// TIA Portal V18 export
DATA_BLOCK "Axis_FB_DB"   // DB2200
// stored: AutoNumber false, InstanceOfName Axis_FB, InstanceOfType FB
"Axis_FB"
   // VAR RETAIN
   //    IAI_Axis { S7_SetPoint := 'True'} : Array[1..3] of "IAI_BASE_FB";
   // END_VAR
BEGIN
   // IAI_Axis[1] : Z轴
   // IAI_Axis[2] : X轴
   // IAI_Axis[3] : Y轴
   // IAI_Axis[1].Par.PosCode : Z轴
   // IAI_Axis[2].Par.PosCode : X轴
   // IAI_Axis[3].Par.PosCode : Y轴
END_DATA_BLOCK
